FUNCTION_BLOCK FB_TagAlarmProps
VAR_INPUT
	sInTimeOcc:STRING[24];
	stInTimeOcc:TIMESTRUCT;
	bInAlarm:BOOL;
	rInturbineStatus:ST_ProcessVariables;
END_VAR
VAR_OUTPUT
	sOutTimeOcc:STRING[24];
	stOutTimeOcc:TIMESTRUCT;
	rOutturbineStatus:ST_ProcessVariables;
END_VAR
VAR
END_VAR

IF bInAlarm THEN
	sOutTimeOcc:=sInTimeOcc;
	stOutTimeOcc:=stInTimeOcc;
	rOutturbineStatus.fFlowSpeed:=rInturbineStatus.fFlowSpeed;
	rOutturbineStatus.fGeneratorSpeed:=rInturbineStatus.fGeneratorSpeed;
	rOutturbineStatus.fPitchAngle:=rInturbineStatus.fPitchAngle;
	rOutturbineStatus.fPower:=rInturbineStatus.fPower;
END_IF

END_FUNCTION_BLOCK

(* stored: Version 1.1.0.1, ProductVersion 3.1.4024.11
   POU FB_TagAlarmProps: Id {24e515fe-b607-4c7c-91fb-668bda84b8a0}, SpecialFunc None *)
